// TIA Portal V17 export
// export: Created 2025-03-10T12:17:22.2259986Z, ExportSetting WithDefaults, DisplayName Totally Integrated Automation Portal, DisplayVersion V17 Update 8, DisplayName TIA Portal Openness, DisplayVersion V17 Update 8, DisplayName TIA Portal Version Control Interface, DisplayVersion V17, DisplayName SINAMICS Startdrive Advanced, DisplayVersion V17 SP2, DisplayName SINAMICS Startdrive G110M, G120, G120C, G120D, G120P, G115D, DisplayVersion V17 SP2, DisplayName SINAMICS Startdrive G130, G150, S120, S150, SINAMICS MV, S210, DisplayVersion V17 SP2, DisplayName STEP 7 Professional, DisplayVersion V17 Update 8, DisplayName SINUMERIK ONE STEP 7 Toolbox, DisplayVersion V17 Update 12, DisplayName SINUMERIK 840D sl STEP 7 Toolbox, DisplayVersion V17 Update 12, DisplayName STEP 7 Safety, DisplayVersion V17 Update 6, DisplayName WinCC Advanced, DisplayVersion V17 Update 8
DATA_BLOCK "DB7236_READ_WRITE_DATA"   // DB7236
{ S7_Optimized_Access := 'FALSE'; DB_Accessible_From_OPC_UA := 'FALSE' }
AUTHOR : ETXETAR
VERSION : 1.0
// stored: AutoNumber false, DBAccessibleFromOPCUA false, DBAccessibleFromWebserver true, IsOnlyStoredInLoadMemory false, IsWriteProtectedInAS false
   VAR RETAIN
      RFID { S7_SetPoint := 'True'} : "READ_WRITE_DATA";
      SAFETY_POSITIONS { S7_SetPoint := 'True'} : "READ_WRITE_DATA";
      ADJUST { S7_SetPoint := 'True'} : "READ_WRITE_DATA";
      ANALOGS { S7_SetPoint := 'True'} : "READ_WRITE_DATA";
      ENABLE_OPTIONS { S7_SetPoint := 'True'} : "READ_WRITE_DATA";
      IO_LINK { S7_SetPoint := 'True'} : "READ_WRITE_DATA";
      MASS_CENTER { S7_SetPoint := 'True'} : "READ_WRITE_DATA";
      FREQUENCY_CONVERTERS { S7_SetPoint := 'True'} : "READ_WRITE_DATA";
      GM_CHIP_CONVEYOR { S7_SetPoint := 'True'} : "READ_WRITE_DATA";
      BK_MIKRO { S7_SetPoint := 'True'} : "READ_WRITE_DATA";
      MEASURE_PROBE { S7_SetPoint := 'True'} : "READ_WRITE_DATA";
      SPINDLES_SET_UP_TWIN { S7_SetPoint := 'True'} : "READ_WRITE_DATA";
      ETXETAR { S7_SetPoint := 'True'} : "READ_WRITE_DATA";
   END_VAR
BEGIN
END_DATA_BLOCK
